// TIA Portal V19 export
TYPE "ValveCtrl"
// stored: Access Published
   STRUCT
      SafeStop : Bool;   // Command: / Emergency stop (device in safe state)
      Rst : Bool;   // Command: / Reset alarms
      MoveRest : Bool;   // Command: / Move to rest command
      MoveWork : Bool;   // Command: / Move to work command
   END_STRUCT;
END_TYPE
